SUBAPPLICATION Uebung_008_AX (* Blinker mit E_CYCLE, E_SWITCH und E_SR *)
  (* Standard: 61499-2; Description: Copyright (c) 2023 Meisterschulen am Ostbahnhof This program and the accompanying materials are made available under the terms of the Eclipse Public License 2.0 which is available at https://www.eclipse.org/legal/epl-2.0/ SPDX-License-Identifier: EPL-2.0 *)
  (* Version 1.0, 2023-10-23, Franz Höpfinger, Meisterschulen am Ostbahnhof, initial API and implementation and/or initial documentation *)
  PACKAGE Uebungen;
  IMPORT logiBUS::io::DQ::logiBUS_DO::Output_Q1;
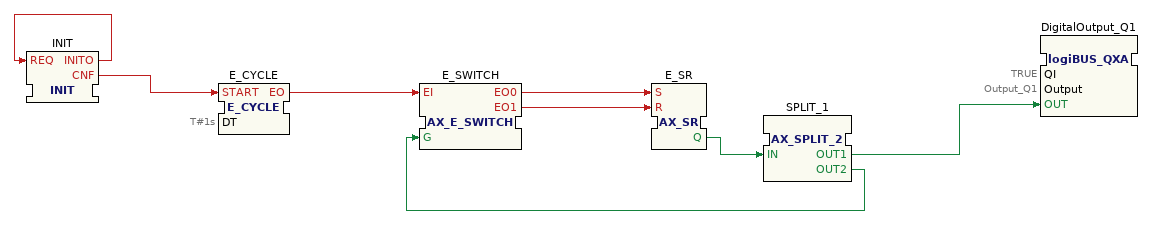
  FBS
    DigitalOutput_Q1 : logiBUS::io::DQ::logiBUS_QXA(QI := TRUE, Output := Output_Q1);
    E_CYCLE : iec61499::events::E_CYCLE(DT := T#1s);
    E_SWITCH : adapter::events::unidirectional::AX_E_SWITCH;
    E_SR : adapter::events::unidirectional::AX_SR;
    INIT : iec61131::booleanOperators::INIT;
    SPLIT_1 : adapter::events::unidirectional::AX_SPLIT_2;
  END_FBS
  EVENT_CONNECTIONS
    E_CYCLE.EO TO E_SWITCH.EI;
    E_SWITCH.EO0 TO E_SR.S;
    E_SWITCH.EO1 TO E_SR.R;
    INIT.INITO TO INIT.REQ;
    INIT.CNF TO E_CYCLE.START;
  END_CONNECTIONS
  ADAPTER_CONNECTIONS
    E_SR.Q TO SPLIT_1.IN;
    SPLIT_1.OUT1 TO DigitalOutput_Q1.OUT;
    SPLIT_1.OUT2 TO E_SWITCH.G;
  END_CONNECTIONS
END_SUBAPPLICATION
